// TIA Portal V17 export
// export: Created 2022-07-16T16:56:10.1206581Z, ExportSetting WithDefaults, DisplayName Totally Integrated Automation Portal, DisplayVersion V17, DisplayName TIA Portal Openness, DisplayVersion V17, DisplayName TIA Portal Version Control Interface, DisplayVersion V17, DisplayName TIA Portal Test Suite Advanced, DisplayVersion V17, DisplayName STEP 7 Professional, DisplayVersion V17, DisplayName STEP 7 Safety, DisplayVersion V17, DisplayName WinCC Professional, DisplayVersion V17
TYPE "methodListType"
// stored: IsFailsafeCompliant false
   STRUCT
      MethodCount { ExternalAccessible := 'False'; ExternalVisible := 'False'; ExternalWritable := 'False'} : UInt;
      ObjectNodes { ExternalAccessible := 'False'; ExternalVisible := 'False'; ExternalWritable := 'False'; S7_SetPoint := 'True'} : Array[0..0] of OPC_UA_NodeId;
      MethodNodes { ExternalAccessible := 'False'; ExternalVisible := 'False'; ExternalWritable := 'False'; S7_SetPoint := 'True'} : Array[0..0] of OPC_UA_NodeId;
      MethodHdls { ExternalAccessible := 'False'; ExternalVisible := 'False'; ExternalWritable := 'False'} : Array[0..0] of DWord;
   END_STRUCT;
   // ObjectNodes[0].NamespaceIndex := 0;
   // ObjectNodes[0].Identifier := WSTRING#'"OPCMethodSetMachineTime_DB"';
   // ObjectNodes[0].IdentifierType := 1;
   // MethodNodes[0].NamespaceIndex := 0;
   // MethodNodes[0].Identifier := WSTRING#'"OPCMethodSetMachineTime_DB".Method';
   // MethodNodes[0].IdentifierType := 1;
END_TYPE
